ABB RobotStudio station: WAAM.rsstnx

Station WAAM (saved by RobotStudio 24.2.10789.0)
Controller IRB4600_45_205, task T_ROB1: task frame (RAPID world) sits at (0, 0, 500) mm in the station
Controller IRB4600_45_205
  mechanical unit ROB_1: IRB4600_45_205_C_01, 6 joints, base frame (0, 0, 0) mm
Layout (positions relative to the parent item):
  - IRB4600_45_205_C_01 [mechanism, from %ABB.RobotStudio.Models.IRB4600%\IRB4600_45_205_C_G_01.rslib] at (0, 0, 500) mm; joint values [0, 0, 0, 0, 0, 0] (rad or m)
  - Fundation [part], size 600 x 600 x 500 mm
  - PieceBase [mechanism] at (-0.06, 0, 0.03) mm
      TCP PieceBase at (616.43, 50, 124) mm, rotated rx 180 ry 0 rz 180 deg
      links: PieceBase
  - WAAM_dispositiv [part] at (1595.69, 0, 0) mm, rotated rx 0 ry 0 rz 90 deg, size 1700 x 1950 x 2110.1 mm
  - IRC5_Single-Cabinet [part, from %ABB.RobotStudio.Models.IRC5%\IRC5_Single-Cabinet.rslib] at (-137.4, -1127.3, 100) mm, rotated rx 90 ry 0 rz -90 deg
  - Fronius_TPS4000_rev0_2 [part, from %ABB.RobotStudio.Models.ArcWelding%\Fronius_TPS4000.rslib] at (2386.57, 495.95, -4.33) mm, rotated rx 0 ry 0 rz 180 deg
  - Gaz [graphiccomponentgroup]
    - Part_3 [part], size 179.4 x 178.8 x 180 mm
    - Part_1 [part], size 180 x 179.6 x 800 mm
  - Gaz_Wire [part], size 2379.8 x 1544.6 x 915 mm
  - AI-IO/v2 [part] at (-257, -82.94, 0) mm, size 200 x 100 x 100 mm
  - IO_cable [part], size 3165.7 x 2417.8 x 109.1 mm
  - PrintedCylinderTool [mechanism] at (0, 0, 0) mm
      TCP PrintedCylinderTool at (162.97, -0.38, 321) mm
      links: piece_tool
Attachment: PieceBase is attached to IRB4600_45_205_C_01 / Link6
Attachment: PrintedCylinderTool is attached to IRB4600_45_205_C_01 / Link6
Targets, tools, work objects and paths stored in the station, written as RAPID:
! task T_ROB1
MODULE user
  PERS tooldata PieceBase:=[TRUE,[[-73.993,0,250.003],[0.707106781,0,-0.707106781,0]],[5,[0,0,1],[1,0,0,0],0,0,0]];
  PERS wobjdata Torch:=[FALSE,TRUE,"ROB_1",[[0,0,0],[1,0,0,0]],[[1937,0,1129.63],[1,0,0,0]]];
  PERS tooldata PrintedCylinderTool:=[TRUE,[[-221,-0.378,187.975],[0.707106781,0,-0.707106781,0]],[5,[0,0,1],[1,0,0,0],0,0,0]];
ENDMODULE

